RoboDK station: GemeloVirtual_DRJ_FINAL.rdk

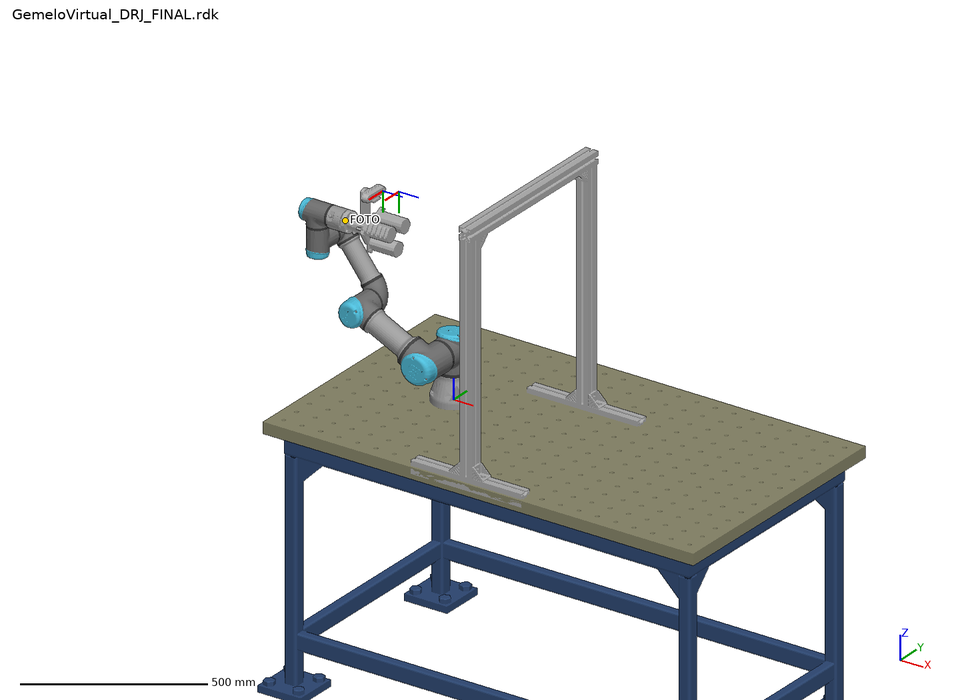
[picture v0: the station drawn from its stored meshes, robots at their saved joint values, targets as dots, program paths as lines]
Station GemeloVirtual_DRJ_FINAL (saved by RoboDK 5.9.2). Poses are relative to the parent item; angles as X-Y-Z fixed-axis rotations.
  - frame UR3e Base at (0, 0, 0) mm
    - robot UR3e: 6 axes, payload 3 kg, reach 500 mm, repeatability 0.03 mm, weight 11 kg
        modified DH rows (alpha deg, a mm, theta deg, d mm): 0, 0, 0, 151.9; 90, 0, 180, 0; 0, 243.55, 0, 0; 0, 213.2, 0, 131.05; -90, 0, 0, 85.35; 90, 0, 180, 92.1
        joint limits [-360, -360, -360, -360, -360, -360] to [360, 360, 360, 360, 360, 360]; home [0, -90, -90, 0, 90, 0]; saved at [-1.86, -24.32, -27.3, -128.19, 91.44, 60]
      - frame Frame 3 at (-105.15, -25.2, 100.11) mm, rotated rx -0.19 ry -0.42 rz -59.99 deg
        - camera Camera 1
      - tool Ensamble_gripper_acoplador, TCP at (0, 0, 0) mm, size 182 x 124.4 x 171 mm, geometry from Ensamble_gripper_acoplador.STEP
    - object Ensamblaje2 at (140, 160, 0) mm, rotated rx 0 ry 0 rz -90 deg, size 590 x 360 x 780 mm, geometry from Ensamblaje2.STEP
    - target FOTO (Cartesian target) at (-266.56, -120.15, 504.99) mm, rotated rx -89.62 ry 59.99 rz -90.09 deg; joints [-1.86, -24.32, -27.3, -128.19, 91.44, 60] of UR3e
    - frame FOTO_FRAME at (-166.57, -90.12, 608.98) mm, rotated rx -90 ry 0 rz -90 deg
      - frame temp_frame at (-74.36, 32.94, -0.01) mm
  - object Table 1400x800x800mm at (0, 0, 0) mm, size 1420 x 820 x 800 mm, geometry from Table-1400x800x800mm.sld
